// TwinCAT 3 PLC project MOCVD_MS
// ProgramVersion: 3.1.4026.14
// libraries:
//   Tc2_ControllerToolbox, * (Beckhoff Automation GmbH)
//   Tc2_ModbusRTU, * (Beckhoff Automation GmbH)
//   Tc2_Standard, * (Beckhoff Automation GmbH)
//   Tc2_System, * (Beckhoff Automation GmbH)
//   Tc2_Utilities, * (Beckhoff Automation GmbH)
// project tree:
//   DUTs/ E_RampGeneratorState.TcDUT (not stored), E_RecipeRun.TcDUT (not stored), E_RecipeRunETMode.TcDUT (not stored), E_TowerLamp.TcDUT (not stored), OperationMode.TcDUT (not stored), outWord.TcDUT (not stored), RampGeneratorInput.TcDUT (not stored), RecipeRunET.TcDUT (not stored), RecipeStep.TcDUT (not stored), ScaleFactor.TcDUT (not stored)
//   FUNCTION/ BOOL_TO_STRING_LHeaterON.TcPOU (not stored), CheckRangeSigned.TcPOU (not stored), CheckRangeUnsigned.TcPOU (not stored), FB_TON_Pausable.TcPOU (not stored), HEXSTR_TO_REAL_LHeaterPV.TcPOU (not stored), Real_To_String_LineHeater.TcPOU (not stored), Real_To_String_ThermalBath.TcPOU (not stored), USINT_TO_WORD_Bit.TcPOU (not stored), WORD_TO_USINT_Bit.TcPOU (not stored)
//   GVLs/ GVL_IO.TcGVL (not stored), RCP.TcGVL (not stored)
//   / PlcTask_Standard.TcTTO
//   POUs/ FB_DeviationCheck.TcPOU (not stored), FB_FaultCheck.TcPOU (not stored), FB_OverLimitCheck.TcPOU (not stored), FB_RampGenerator.TcPOU (not stored), FB_RampGenerator_1.TcPOU, FB_RecipeSequencer.TcPOU (not stored), FB_SensorLimitCheck.TcPOU (not stored), FB_TON_Pausable_1.TcPOU, F_ResetTimersAndRCPTimes.TcPOU (not stored), MAIN.TcPOU (not stored), P11_E3508.TcPOU (not stored), P12_IQ_PLUS.TcPOU (not stored), P13_LineHeater.TcPOU (not stored), P14_ThermalBath.TcPOU (not stored), P15_RotationOperation.TcPOU (not stored), P16_CoverOperation.TcPOU (not stored), P17_DOROperation.TcPOU (not stored), P20_BackgroundCom.TcPOU (not stored), P21_Background_LineHeater.TcPOU (not stored), P22_Background_ThermalBath.TcPOU (not stored), P30_ManualControl.TcPOU (not stored), P50_RecipeControl.TcPOU (not stored), P70_Interface.TcPOU (not stored), P90_Interlock.TcPOU (not stored), P91_Monitoring.TcPOU (not stored), P92_Maintenance.TcPOU (not stored)
// real-time tasks:
//   TASK PlcTask_Standard: cycle T#10ms, priority 21, ADS port 350
//   TASK PlcTask: cycle T#2ms, priority 19, ADS port 351
// I/O:
//   DEVICE Device 1 (EtherCAT) (disabled), AmsNetId 211.225.0.130.2.1
//     Term 1 (EK1200) [EK1200-5000 EtherCAT Power supply (2A E-Bus)]
//       Term 2 (EL6752) [EL6752 DeviceNet Master]
//       Term 3 (EL9011) [EL9011 End Terminal]
//   DEVICE Device 2 (EL6752) (disabled), AmsNetId 10.10.10.10.3.1
//     Box 1  (BK5220) // Bus Coupler
//     Box 2  (BK5220) // Bus Coupler
//     N4E0 1 // EDS-File: 'OPP6-2D.eds' DescText: OPP6-2D Vendor: CKD Corporation Device Type: Generic Device Product Name: OPP6-2D Catalog Number:
//     N4E0 2 // EDS-File: 'OPP6-2D.eds' DescText: OPP6-2D Vendor: CKD Corporation Device Type: Generic Device Product Name: OPP6-2D Catalog Number:
//     IQ-Plus // EDS-File: 'TBJQPDNG-L041X01 155Out154.eds' DescText: Intellisys IQ-Plus Vendor: Nor-Cal Products Device Type: Process Control Valve Product Name: INTELLISYS Catalog Number: IQ-Plus
//     E3508 // EDS-File: '3500-3.eds' DescText: Eurotherm 3500 Vendor: Eurotherm Device Type: Generic Product Name: Eurotherm 3500 Catalog Number:
//   DEVICE Device 3 (NOV-DP-RAM) (disabled)

CONFIGURATION MOCVD_MS
    RESOURCE PLC ON TwinCAT3
        TASK PlcTask_Standard(INTERVAL := T#10ms, PRIORITY := 21);
        PROGRAM MAIN WITH PlcTask_Standard : MAIN;
    END_RESOURCE
END_CONFIGURATION

// ---- POUs/FB_RampGenerator_1.TcPOU
FUNCTION_BLOCK FB_RampGenerator_1
VAR_INPUT
	//bStart_Stop			: BOOL := TRUE;
	//bAlarmReset			: BOOL;
	rInitValue		: REAL;
	rTargetValue	: REAL;
	nRampTime		: INT := 1; // Second
	nState			: INT; //0:Init State
END_VAR

VAR_OUTPUT
	rControlValue	: LREAL;
	rStartValue		: REAL;
END_VAR

VAR
	// for FB_CTRL_RAMP_GENERATOR Variable
	(* input *)
	bEnable			: BOOL; // Reference
	(* output *)
	bValueReached	: BOOL;
	(* function block *)
	fbCTRL_RAMP_GENERATOR			: FB_CTRL_RAMP_GENERATOR;
	stCTRL_RAMP_GENERATOR_PARAMS	: ST_CTRL_RAMP_GENERATOR_PARAMS;
	eErrorId						: E_CTRL_ERRORCODES;
	bError							: BOOL;
	bInit							: BOOL := TRUE;
	(* Operation Parameter*)
	rRampingRatio			: REAL;		
END_VAR

(* Convert to Normalization, Ramp Valve Calculation*)
IF nRampTime = 0 THEN
	bEnable := FALSE;
ELSE
	rRampingRatio := ABS(rTargetValue - rStartValue) / nRampTime * 0.1; //Second
END_IF

CASE nState OF
	0: // Init Sate
		rStartValue := rInitValue;
		bInit := TRUE;
		bValueReached := TRUE;
	10: // RUN
		IF (rTargetValue > 0) OR (rStartValue > 0) THEN
			bEnable := TRUE;
			bInit := TRUE;
		ELSE
			bEnable := FALSE;
			bInit := FALSE;
		END_IF
// 	20: //PAUSE
// 		bEnable := TRUE;
// 	30: //RESTART
// 		bEnable := TRUE;	
// 	40: //STOP
// 		bEnable := FALSE;
// 		bInit := TRUE;
// 		bValueReached := TRUE;
// 	50: //END
// 		bEnable := FALSE;
// 		bInit := TRUE;
// 		bValueReached := TRUE;

END_CASE

IF bInit THEN
	(* init parameter struct *)
	stCTRL_RAMP_GENERATOR_PARAMS.tTaskCycleTime		:= T#100MS;
	stCTRL_RAMP_GENERATOR_PARAMS.tCtrlCycleTime		:= T#100MS;
	stCTRL_RAMP_GENERATOR_PARAMS.fVeloPos			:= rRampingRatio; (* in units per second *)
	stCTRL_RAMP_GENERATOR_PARAMS.fVeloNeg			:= rRampingRatio; (* in units per second *)
	(* reset the init flag *)
	bInit := FALSE;
END_IF

IF rTargetValue <> rStartValue THEN
	(* call function block *)
	fbCTRL_RAMP_GENERATOR(
		bEnable			:= bEnable,
		fStart			:= rStartValue,
		fTarget			:= rTargetValue,
		stParams		:= stCTRL_RAMP_GENERATOR_PARAMS,
		fOut			=> rControlValue,
		bValueReached	=> bValueReached,
		bError			=> bError,
		eErrorId		=> eErrorId);
ELSE
	fbCTRL_RAMP_GENERATOR.bEnable := FALSE;
END_IF

IF bValueReached THEN
	rStartValue := LREAL_TO_REAL(rControlValue);
END_IF

(* Convert to Writing Value *)
//nControlValue := REAL_TO_INT(rControlValue);

END_FUNCTION_BLOCK

// ---- POUs/FB_TON_Pausable_1.TcPOU
FUNCTION_BLOCK FB_TON_Pausable_1
VAR_INPUT
	IN      : BOOL;     (* Start/Stop the timer *)
    PT      : TIME;     (* Preset time *)
    PAUSE   : BOOL;     (* Pause the timer *)
END_VAR
VAR_OUTPUT
	Q       : BOOL;     (* Output: TRUE when PT is reached *)
    ET      : TIME;     (* Elapsed time *)
END_VAR
VAR
	// Internal variables
    fbTON   : TON;      (* Standard TON to do the actual timing when not paused *)
    tElapsedAtPause : TIME; (* Stores ET when paused *)
    bWasPaused      : BOOL; (* Helps detect the rising edge of PAUSE *)
    bOldIn          : BOOL; (* Stores previous IN state for rising/falling edge detection *)
END_VAR

IF NOT IN THEN
    // Reset condition: IN is FALSE
    tElapsedAtPause := T#0S;
    ET := T#0S;
    Q := FALSE;
    fbTON(IN := FALSE); // Ensure internal TON is also reset
    bWasPaused := FALSE; // Reset pause state
ELSIF IN THEN
    // Timer is active
    IF PAUSE THEN
        // PAUSE is active
        IF NOT bWasPaused THEN
            // Rising edge of PAUSE: Capture current elapsed time from TON
            tElapsedAtPause := tElapsedAtPause + fbTON.ET;
            bWasPaused := TRUE;
        END_IF
        // Timer is paused: ET does not advance
        ET := tElapsedAtPause;
        Q := (ET >= PT); // Q remains based on the paused ET
        fbTON(IN := FALSE); // Stop the internal TON from running
    ELSE (* NOT PAUSE *)
        // PAUSE is not active, run the timer
        bWasPaused := FALSE; // Clear paused state

        // Adjust PT for the internal TON to account for time spent paused
        // Only call TON if IN is TRUE and NOT PAUSE
        fbTON(
            IN := TRUE,
            PT := PT - tElapsedAtPause (* Subtract time already elapsed/paused *)
        );

        // Calculate actual ET for output
        // It's the time accumulated before pause + time accumulated after resume
        ET := tElapsedAtPause + fbTON.ET;
        Q := fbTON.Q;
    END_IF
END_IF

// Store current IN state for next cycle's edge detection
bOldIn := IN;

END_FUNCTION_BLOCK
